// TIA Portal V20 export
FUNCTION_BLOCK "FB_McpKeysSignals"   // FB422, SCL
{ S7_Optimized_Access := 'TRUE' }
// stored: AutoNumber false, MemoryReserve 100, SetENOAutomatically false
   VAR_INPUT
      iKeyHWStatus { ExternalAccessible := 'False'; ExternalVisible := 'False'; ExternalWritable := 'False'} : Bool;   // PLC Digital Input Hardware status
   END_VAR
   VAR_OUTPUT
      oLedHWStatus : Bool;
   END_VAR
   VAR
      sKeySWStatus : Bool;
      sKeySWToggleStatus : Bool;
      sKeyDisable : Bool;
      sKeySWPositiveFront : Bool;
      sKeySWNegativeFront : Bool;
      sKeySWTogglePositiveFront : Bool;
      sKeySWToggleNegativeFront : Bool;
      sLedSWStatus : Bool;
      sRT_KeySWPositiveFront { S7_SetPoint := 'True'} : R_TRIG;
      sFT_KeySWNegativeFront { S7_SetPoint := 'True'} : F_TRIG;
      sRT_KeySWTogglePositiveFront { S7_SetPoint := 'True'} : R_TRIG;
      sFT_KeySWToggleNegativeFront { S7_SetPoint := 'True'} : F_TRIG;
   END_VAR
BEGIN
   REGION Description header 
       //==================================================================================
       // POSALUX Swiss SA / (C) Copyright 2025
       //----------------------------------------------------------------------------------
       // Title: Management of inputs and outputs for MCP and external buttons 
       // Comment/Function: 
       //
       // Author: Fabien Waldt
       // Engineering: TIA Portal v19
       //----------------------------------------------------------------------------------
       // Change log table:
       // Version  | Date     | Expert in charge | Changes applied
       // ---------|----------|------------------|------------------------------------
       // 00.00.01 | 20250911 | WFA              | First released version
       // 00.00.02 | 20260218 | WFA              | Remove reset toggle when disable
       // ==================================================================================
   END_REGION

   REGION Inputs keys
           // Management of inputs for each customerkey MCP button 
           // Management of the software input
            IF NOT #sKeyDisable THEN
                #sKeySWStatus := #iKeyHWStatus;
            END_IF;

           // Rising/falling edge detection when pressing the button
           #sRT_KeySWPositiveFront(CLK := #sKeySWStatus,
                                  Q => #sKeySWPositiveFront);

           #sFT_KeySWNegativeFront(CLK := #sKeySWStatus,
                                  Q => #sKeySWNegativeFront);

           // Toggle state update
           IF #sKeySWPositiveFront  THEN
               #sKeySWToggleStatus := NOT #sKeySWToggleStatus;
           END_IF;

           // Rising/falling edge detection of the toggle state
           #sRT_KeySWTogglePositiveFront(CLK := #sKeySWToggleStatus,
                                        Q => #sKeySWTogglePositiveFront);

           #sFT_KeySWToggleNegativeFront(CLK := #sKeySWToggleStatus,
                                        Q => #sKeySWToggleNegativeFront);
   END_REGION

   REGION Outputs LED   
       #oLedHWStatus := #sLedSWStatus;
   END_REGION
END_FUNCTION_BLOCK
